{attribute 'qualified_only'}
VAR_GLOBAL
	// Pitch Mechanism
	{attribute 'TcLinkTo' := '.diEncCnt:=TIIB[EL5042_M2L0_PitchBender]^FB Inputs Channel 1^Position'}
	M2L0_Pitch : HOMS_PitchMechanism := (ReqPosLimHi := 154.9,
		                                 ReqPosLimLo := -45.1,
		                                 diEncPosLimHi := 9550777,
		                                 diEncPosLimLo := 9448178);
    // M2L0 Flow Press Sensors
    {attribute 'TcLinkTo' := '.iRaw := TIIB[EL3054_M2L0_FLOW_PRESS]^AI Standard Channel 1^Value'}
    fM2L0_Flow_1 : FB_AnalogInput;
    {attribute 'pytmc' := '
		pv: MR2L0:HOMS:FLOW:1
        field: EGU lpm
        io: i
    '}   
    fM2L0_Flow_1_val : LREAL;
    {attribute 'TcLinkTo' := '.iRaw := TIIB[EL3054_M2L0_FLOW_PRESS]^AI Standard Channel 2^Value'}
    fM2L0_Flow_2 : FB_AnalogInput;
    {attribute 'pytmc' := '
		pv: MR2L0:HOMS:FLOW:2
        field: EGU lpm
        io: i
    '} 
    fM2L0_Flow_2_val : LREAL; 
    {attribute 'TcLinkTo' := '.iRaw := TIIB[EL3054_M2L0_FLOW_PRESS]^AI Standard Channel 3^Value'}
    fM2L0_Press_1 : FB_AnalogInput;
    {attribute 'pytmc' := '
		pv: MR2L0:HOMS:PRESS:1
        field: EGU bar
        io: i
    '}      
    fM2L0_Press_1_val : LREAL;
END_VAR

(* stored: Version 1.1.0.1, ProductVersion 3.1.4022.18
   GVL GVL_M2L0: Id {b4287d9d-45c2-46f6-b4bf-11d58d75255d} *)
